FUNCTION_BLOCK MiscHandling
VAR_INPUT
END_VAR
VAR_OUTPUT
END_VAR
VAR
	// Digital Probe Trigger output to Pin 29 of PC
	PCProbeOutput AT %Q*: BOOL := FALSE;
	// Digital Probe Input (Normally Closed)
	ProbeInput AT %I*: BOOL := TRUE;
	// Air Pressure >90psi signal to PC Pin 10
	PCPressureOutput AT %Q*: BOOL := FALSE;
	// Air Pressure >90psi signal from sensor
	PressureSensorInput AT %I*: BOOL := FALSE;
END_VAR

PCProbeOutput := NOT ProbeInput;
PCPressureOutput := PressureSensorInput;

END_FUNCTION_BLOCK

(* stored: Version 1.1.0.1, ProductVersion 3.1.4022.12
   POU MiscHandling: Id {7703155d-3f80-4f64-a8fb-b20c126e77fb}, SpecialFunc None *)
